(* CODESYS project udp_sample190212.1.project

Project tree, tasks and I/O mapping:
  Device : Changsha Xiangji-ARM Cortex A9(xilinx zynq7000)-linux, Changsha Xiangji Hiden Technology Co.Ltd, version 3.5.10.40
    application Application
      libraries: Standard, * (System); CAA Types Extern, * (CAA Technical Workgroup); CAA File, * (CAA Technical Workgroup); CAA DTUtil Extern, * (CAA Technical Workgroup); Cyber Udp Library, 3.5.12.40 (Cyber Company)
      task MainTask (cyclic, interval 10 ms, priority 1) calls PLC_PRG
      program PLC_PRG [ST]
      global variables GVL
    SoftMotion General Axis Pool
*)

// Device/Application/GVL
{attribute 'qualified_only'}
VAR_GLOBAL
	iccid :STRING;
	lac :UINT;
	cid :UINT;
	sn :STRING;
	work_time :UDINT;
END_VAR

// Device/Application/PLC_PRG
PROGRAM PLC_PRG
VAR
	is_inited :BOOL := FALSE;
	
	udp_handle :CAA.HANDLE; 
	udp_init_fb:Udp_Init;
	udp_write_fb:Udp_Write;
	udp_read_fb:Udp_Read;


	size :CAA.SIZE;	
	Writebuffer: 			ARRAY[1..200] OF BYTE;
	Readbuffer: 			ARRAY[1..10] OF BYTE;
	ReadbufferStr: STRING;
	atcState :INT := 0;
	
	writeUdpState :INT := 0;
	readUdpState :INT := 0;
	
	i :INT;
	count :INT := 0;
	
	rtc_fb: RTC;
	dtu_set_dt_fb: dtu.SetDateAndTime;
	
	sn_file_name :STRING := 'sn.txt';
	time_file_name :STRING := 'r_mins.txt';
	is_read :BOOL := FALSE;
	read_count :INT := 0;
	readFileState :INT := 0;
	ton01 :TON;
END_VAR


IF NOT is_inited THEN
	udp_init_fb(ip_addr := '47.107.240.29', port := 23457);
	IF udp_init_fb.init_mode = 1 THEN
		is_inited := TRUE;
		udp_handle := udp_init_fb.udp_handle;
	END_IF
END_IF

IF NOT is_inited THEN  //没有初始化完成,直接返回
	RETURN;
END_IF

CASE atcState OF
	0:  //发送数据
		// if error, atcState return 32767, if done, atcState return 1
		udp_write_fb(com := udp_handle, buffer:= ADR(Writebuffer), size := 21);
		IF udp_write_fb.atcState = 1 THEN
			atcState := 10;
		END_IF	
	10:  //延时50ms，等待服务器回复
		ton01(in := TRUE, PT := TIME#50MS);
		IF ton01.Q THEN
			ton01(in := FALSE);
			atcState := 20;
		END_IF
	20:  //接收数据
		// if error, atcState return 32767, if done, atcState return 1
		udp_read_fb(com:= udp_handle, buffer:= ADR(Readbuffer), rsize := SIZEOF(Readbuffer));
		IF udp_read_fb.atcState = 1 THEN
			atcState := 30;
		END_IF
	30:  //延时2S，再发下一帧
		ton01(in := TRUE, PT := TIME#2S);
		IF ton01.Q THEN
			ton01(in := FALSE);
			atcState := 0;
		END_IF	
END_CASE

END_PROGRAM
